FUNCTION_BLOCK EK1100

VAR_INPUT
    En              : BOOL;
    iTerminal_ID    : INT;
    ErrorSystem     : POINTER TO ST_ErrorSystem;
END_VAR

VAR_OUTPUT
    EnO     : BOOL;
    bError  : BOOL;
END_VAR

VAR
    InfoData_State  AT %I*  : UINT;

    //FB-s
    EK1100_Error    : FB_TerminalError;
END_VAR

(*
* TODO: DONE!
*)
EnO:=En;

//Error FB instance
EK1100_Error(
    En                  := TRUE,
    iTerminal_ID        := iTerminal_ID,
    bWcState            := FALSE,
    uiInfoData_State    := InfoData_State,
    pErrorSystem        := ErrorSystem,
    bError              => bError,
);

END_FUNCTION_BLOCK

(* stored: Version 1.1.0.1, ProductVersion 3.1.4024.0
   POU EK1100: Id {658f73e7-ff3e-4539-b62c-4f4914e2b326}, SpecialFunc None *)
